PROGRAM pouMcPrompts
VAR
	


idbMsgPrompt: FB_CheckMessageBounds;
	sdfsdf: BOOL;
	msgPowerON: BOOL;
	test: BOOL;
END_VAR

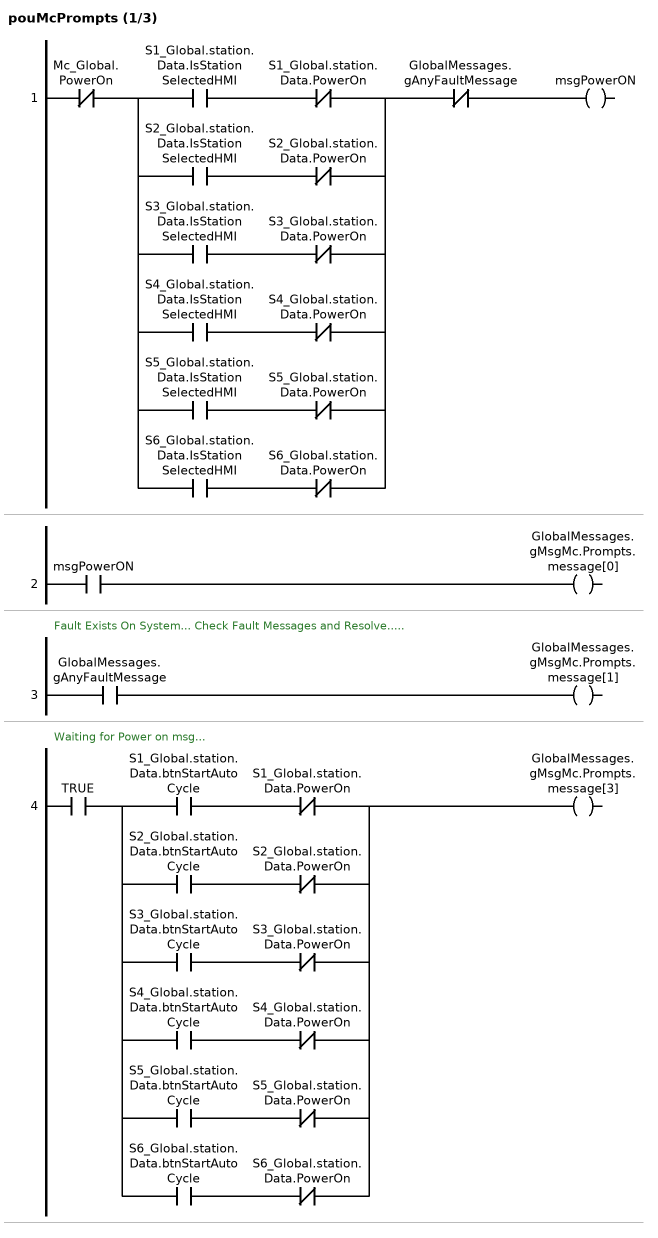
// NETWORK 1
msgPowerON := NOT Mc_Global.PowerOn AND (S1_Global.station.Data.IsStationSelectedHMI AND NOT S1_Global.station.Data.PowerOn OR S2_Global.station.Data.IsStationSelectedHMI AND NOT S2_Global.station.Data.PowerOn OR S3_Global.station.Data.IsStationSelectedHMI AND NOT S3_Global.station.Data.PowerOn OR S4_Global.station.Data.IsStationSelectedHMI AND NOT S4_Global.station.Data.PowerOn OR S5_Global.station.Data.IsStationSelectedHMI AND NOT S5_Global.station.Data.PowerOn OR S6_Global.station.Data.IsStationSelectedHMI AND NOT S6_Global.station.Data.PowerOn) AND NOT GlobalMessages.gAnyFaultMessage;

// NETWORK 2
GlobalMessages.gMsgMc.Prompts.message[0] := msgPowerON;

// NETWORK 3
// Fault Exists On System... Check Fault Messages and Resolve.....
GlobalMessages.gMsgMc.Prompts.message[1] := GlobalMessages.gAnyFaultMessage;

// NETWORK 4
// Waiting for Power on msg...
GlobalMessages.gMsgMc.Prompts.message[3] := TRUE AND (S1_Global.station.Data.btnStartAutoCycle AND NOT S1_Global.station.Data.PowerOn OR S2_Global.station.Data.btnStartAutoCycle AND NOT S2_Global.station.Data.PowerOn OR S3_Global.station.Data.btnStartAutoCycle AND NOT S3_Global.station.Data.PowerOn OR S4_Global.station.Data.btnStartAutoCycle AND NOT S4_Global.station.Data.PowerOn OR S5_Global.station.Data.btnStartAutoCycle AND NOT S5_Global.station.Data.PowerOn OR S6_Global.station.Data.btnStartAutoCycle AND NOT S6_Global.station.Data.PowerOn);

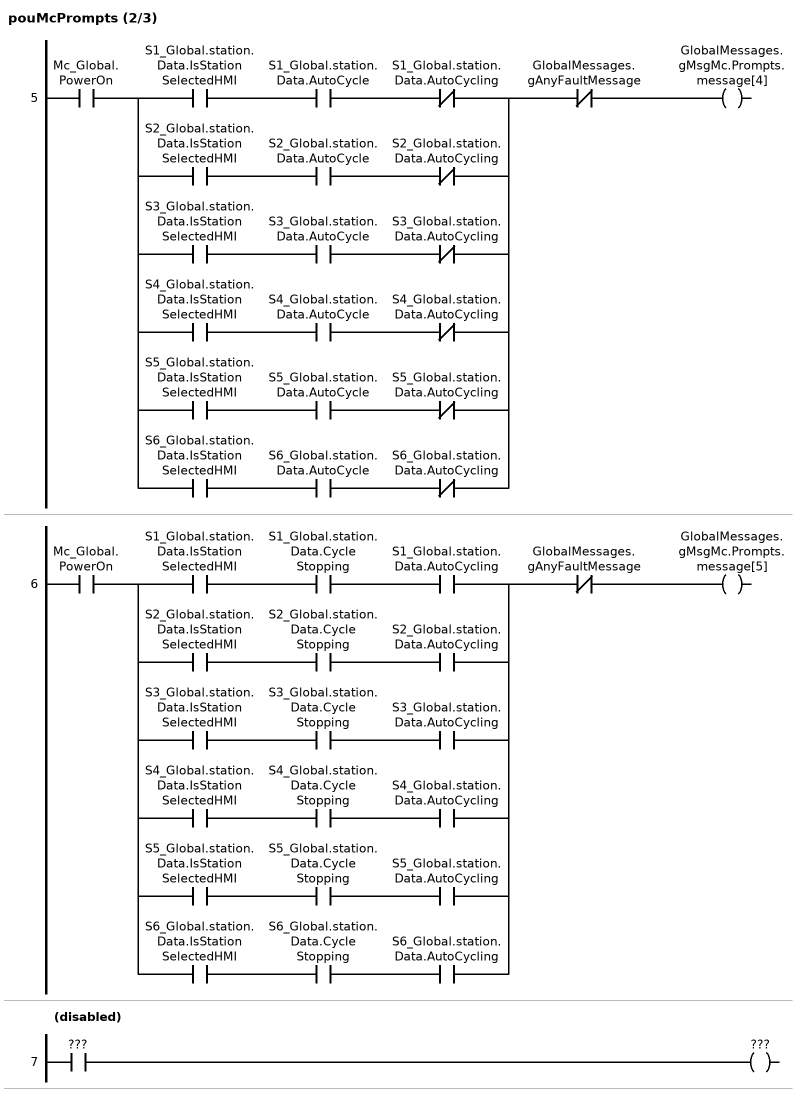
// NETWORK 5
GlobalMessages.gMsgMc.Prompts.message[4] := Mc_Global.PowerOn AND (S1_Global.station.Data.IsStationSelectedHMI AND S1_Global.station.Data.AutoCycle AND NOT S1_Global.station.Data.AutoCycling OR S2_Global.station.Data.IsStationSelectedHMI AND S2_Global.station.Data.AutoCycle AND NOT S2_Global.station.Data.AutoCycling OR S3_Global.station.Data.IsStationSelectedHMI AND S3_Global.station.Data.AutoCycle AND NOT S3_Global.station.Data.AutoCycling OR S4_Global.station.Data.IsStationSelectedHMI AND S4_Global.station.Data.AutoCycle AND NOT S4_Global.station.Data.AutoCycling OR S5_Global.station.Data.IsStationSelectedHMI AND S5_Global.station.Data.AutoCycle AND NOT S5_Global.station.Data.AutoCycling OR S6_Global.station.Data.IsStationSelectedHMI AND S6_Global.station.Data.AutoCycle AND NOT S6_Global.station.Data.AutoCycling) AND NOT GlobalMessages.gAnyFaultMessage;

// NETWORK 6
GlobalMessages.gMsgMc.Prompts.message[5] := Mc_Global.PowerOn AND (S1_Global.station.Data.IsStationSelectedHMI AND S1_Global.station.Data.CycleStopping AND S1_Global.station.Data.AutoCycling OR S2_Global.station.Data.IsStationSelectedHMI AND S2_Global.station.Data.CycleStopping AND S2_Global.station.Data.AutoCycling OR S3_Global.station.Data.IsStationSelectedHMI AND S3_Global.station.Data.CycleStopping AND S3_Global.station.Data.AutoCycling OR S4_Global.station.Data.IsStationSelectedHMI AND S4_Global.station.Data.CycleStopping AND S4_Global.station.Data.AutoCycling OR S5_Global.station.Data.IsStationSelectedHMI AND S5_Global.station.Data.CycleStopping AND S5_Global.station.Data.AutoCycling OR S6_Global.station.Data.IsStationSelectedHMI AND S6_Global.station.Data.CycleStopping AND S6_Global.station.Data.AutoCycling) AND NOT GlobalMessages.gAnyFaultMessage;

// NETWORK 7 (disabled)
// ??? := ???;

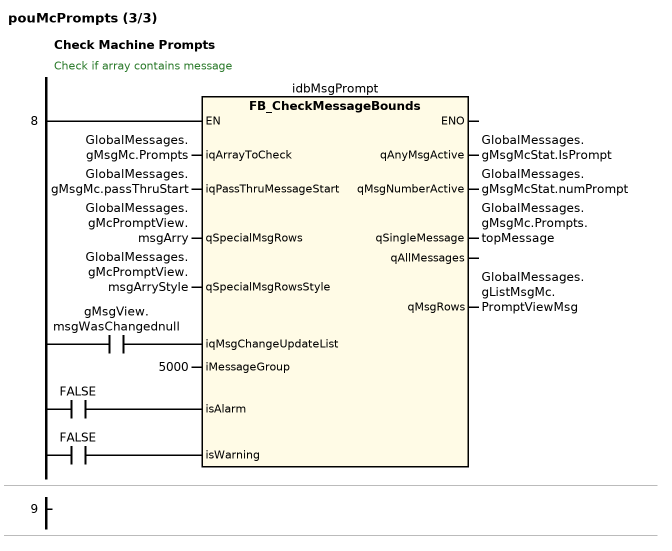
// NETWORK 8: Check Machine Prompts
// Check if array contains message
idbMsgPrompt(
    iqArrayToCheck := GlobalMessages.gMsgMc.Prompts,
    iqPassThruMessageStart := GlobalMessages.gMsgMc.passThruStart,
    qSpecialMsgRows := GlobalMessages.gMcPromptView.msgArry,
    qSpecialMsgRowsStyle := GlobalMessages.gMcPromptView.msgArryStyle,
    iqMsgChangeUpdateList := gMsgView.msgWasChangednull,
    iMessageGroup := 5000,
    isAlarm := FALSE,
    isWarning := FALSE,
    qAnyMsgActive => GlobalMessages.gMsgMcStat.IsPrompt,
    qMsgNumberActive => GlobalMessages.gMsgMcStat.numPrompt,
    qSingleMessage => GlobalMessages.gMsgMc.Prompts.topMessage,
    qMsgRows => GlobalMessages.gListMsgMc.PromptViewMsg); // FB_CheckMessageBounds

// NETWORK 9

END_PROGRAM

(* stored: Version 1.1.0.1, ProductVersion 3.1.4024.11
   POU pouMcPrompts: Id {d586c653-4092-490f-b1fa-a2659fd64310}, SpecialFunc None *)
